// TIA Portal V19 export
FUNCTION_BLOCK "TYPIC_C301_SF_VEN"   // FB6, FBD
TITLE = TYPIC_C301_SF_VEN: Ventilator verkeerskoker
{ S7_Optimized_Access := 'TRUE' }
AUTHOR : OCOTECH
FAMILY : Typical
NAME : C301.803
// Logisch Object Besturing: C301.803
// 
// De subfunctie “ventilator verkeerskoker” verzorgt de bediening en sturing van een ventilator vanuit 3B en is tevens het raakvlak tussen 3B en de interne sturing van de ventilator.
// 
// De subfunctie kan zowel gebruikt worden voor langsventilatoren als ingangsventilatoren.
// 
// Een langsventilator heeft 2 mogelijke draairichtingen:
//  Rijrichting
//  Tegenrij
// 
// Een ingangsventilator heeft slechts 1 mogelijke draairichting:
//  Rijrichting
// 
// Deze typical werkt op dezelfde manier voor ingangsventilatoren als langsventilatoren. Bij ingangsventilatoren komen in de praktijk een aantal mogelijkheden nooit voor:
//  Op IRIS SCADA is er een andere typical voor ingangsventilatoren, deze typical heeft geen mogelijkheid voor bediening “Tegenrij”
//  Vanuit de basisfunctie wordt een cluster met ingangsventilatoren nooit in “Tegenrij” aangestuurd 
//  De waarde “Tegenrij” is nooit van toepassing voor statussen of sturingen
//  Signaleringen met betrekking tot “Tegenrij” komen nooit op
// stored: MemoryReserve 10, SetENOAutomatically false
   VAR_INPUT
      CFG_PWR { ExternalAccessible := 'False'; ExternalVisible := 'False'; ExternalWritable := 'False'} : Real;   // Vermogen ventilator
      CFG_IVEN { ExternalAccessible := 'False'; ExternalVisible := 'False'; ExternalWritable := 'False'} : USInt;   // De ventilator is een ingangsventilator
      STU_CMD_AUT { ExternalAccessible := 'False'; ExternalVisible := 'False'; ExternalWritable := 'False'} : USInt;   // Groepscommando: schakel in automatisch
      STU_ALG_LCK_SIG { ExternalAccessible := 'False'; ExternalVisible := 'False'; ExternalWritable := 'False'} : USInt;   // Onderdruk alarmen
      STU_ENE_VGV_AAN { ExternalAccessible := 'False'; ExternalVisible := 'False'; ExternalWritable := 'False'} : USInt;   // Vrijgeven of verhinderen bijschakelen energieverbruikers (verlichting / ventilatie)
   END_VAR
   VAR_OUTPUT
      VAR_VEN { ExternalAccessible := 'False'; ExternalVisible := 'False'; ExternalWritable := 'False'} : "C301_VAR_VEN_TYPIC";   // Struct met alle variabelen van de ventilator
      STU_IF_VEN { ExternalAccessible := 'False'; ExternalVisible := 'False'; ExternalWritable := 'False'} : "C301_STU_IF_VEN_TYPIC";   // Struct met alle sturingen naar de functie (IF) in de interne sturing van de ventilator
   END_VAR
   VAR_IN_OUT
      CMD : USInt;   // Sturing ventilator
      BST : USInt;   // Sturing In Dienst / Uit Dienst
      VGV_BEV : USInt;   // Vrijgave ventilator-beveiligingen onbalans en temperatuur
   END_VAR
   VAR
      BED : Struct   // Bedieningen
         ALG : Struct   // Gewenste stand
            X : "UDT_BED_ALG";
            KNOP { S7_SetPoint := 'True'} : Array[0..3] of "UDT_BED_KNOP";
         END_STRUCT;
         BST : Struct   // Bestuurbaarheid
            X : "UDT_BED_ALG";
            KNOP { S7_SetPoint := 'True'} : Array[0..1] of "UDT_BED_KNOP";
         END_STRUCT;
         RES : Struct   // Reset Storingen
            X : "UDT_BED_ALG";
            KNOP { S7_SetPoint := 'True'} : Array[0..0] of "UDT_BED_KNOP";
         END_STRUCT;
      END_STRUCT;
      BED_ALG { ExternalWritable := 'False'} : "TYPIC_HF_BED_ALG_KNOP";   // Gewenste stand
      BED_BST { ExternalWritable := 'False'} : "TYPIC_HF_BED_ALG_KNOP";   // Bestuurbaarheid
      BED_RES { ExternalWritable := 'False'} : "TYPIC_HF_BED_ALG_KNOP";   // Reset Storingen
      SIG { ExternalWritable := 'False'} : Struct   // Signaleringen
         AA01 : Bool;   // Ventilator niet bestuurbaar
         AA02 : Bool;   // Ventilator geeft storing, maar is bestuurbaar
         A001 : Bool;   // Beveiliging aangesproken
         A002 : Bool;   // Algemene storing MCC
         A003 : Bool;   // Te hoge temperatuur in de wikkelingen van de motor van de ventilator
         A004 : Bool;   // De ventilator is in onbalans
         A005 : Bool;   // Fout stroommeting fase 1
         A006 : Bool;   // Fout stroommeting fase 2
         A007 : Bool;   // Fout stroommeting fase 3
         A008 : Bool;   // Motorlade uitgeschakeld
         A009 : Bool;   // Motorlade in test
         A010 : Bool;   // Motorlade uitgereden
         A011 : Bool;   // Draadbreuk trillingsmeting
         A012 : Bool;   // Meetbereik trillingsmeting overschreden
         AT01 : Bool;   // Foute terugmelding: Motor aangestuurd, terugmelding Aan niet (of te laat) ontvangen
         AT02 : Bool;   // Foute terugmelding: Motor niet aangestuurd, terugmelding Aan blijft aanwezig
         AT03 : Bool;   // Foute terugmeldingen: terugmeldingen Positief en negatief tegelijkertijd
         M001 : Bool;   // Werkschakelaar uitgeschakeld
      END_STRUCT;
      VAR { ExternalWritable := 'False'} : Struct   // Variabelen
         TYD_TOT_AAN_UUR : USInt;   // Totaal aantal draaiuren
         ENE_MWA1 : Real;   // Stroommeting fase 1
         ENE_MWA2 : Real;   // Stroommeting fase 2
         ENE_MWA3 : Real;   // Stroommeting fase 3
         TRL_MWA : USInt;   // Trillingsmeting
         RNB : USInt;   // Reden niet bestuurbaar
         AUT : USInt;   // Beveiliging aangesproken
         VGV_SIG_VOP : Bool;   // TRUE = Signaleringen vrijgegeven voor verkeersoperator FALSE = Onderdrukt
         STS : USInt;   // Status van de ventilator
         DIR : USInt;   // Richting van de ventilator
         BMO : USInt;   // Bedieningsmode
         BST { ExternalAccessible := 'False'; ExternalVisible := 'False'} : USInt;   // Bestuurbaarheid
         PWR { ExternalAccessible := 'False'; ExternalVisible := 'False'} : Real;   // Vermogen van de ventilator
         TYD_TOT_AAN { ExternalAccessible := 'False'; ExternalVisible := 'False'} : USInt;   // Totaal aantal draaiuren
      END_STRUCT;
      HF_BST_OBS { ExternalAccessible := 'False'; ExternalVisible := 'False'; ExternalWritable := 'False'} : "TYPIC_HF_BST_OBS";   // Hulp functie besturing
   END_VAR
   // // BED.ALG.KNOP[0] : Auto
   // // BED.ALG.KNOP[1] : Rijrichting
   // // BED.ALG.KNOP[2] : Tegenrij
   // // BED.ALG.KNOP[3] : Uit
   // // BED.BST.KNOP[0] : InDienst
   // // BED.BST.KNOP[1] : UitDienst
   // // BED.RES.KNOP[0] : Reset
BEGIN

REGION Network 1: START
END_REGION

REGION Network 2: +++ Bedieningen +++
   // Vrijgave en verwerking van de bedieningen (centrale en lokale bediening). De bedienwaardes worden daarna in de verdere deelfunctionaliteiten gebruikt.
END_REGION

REGION Network 3: Knoppen BED_ALG(Gewenste stand)
   // Waardes en vrijge van de knoppen BED_ALG
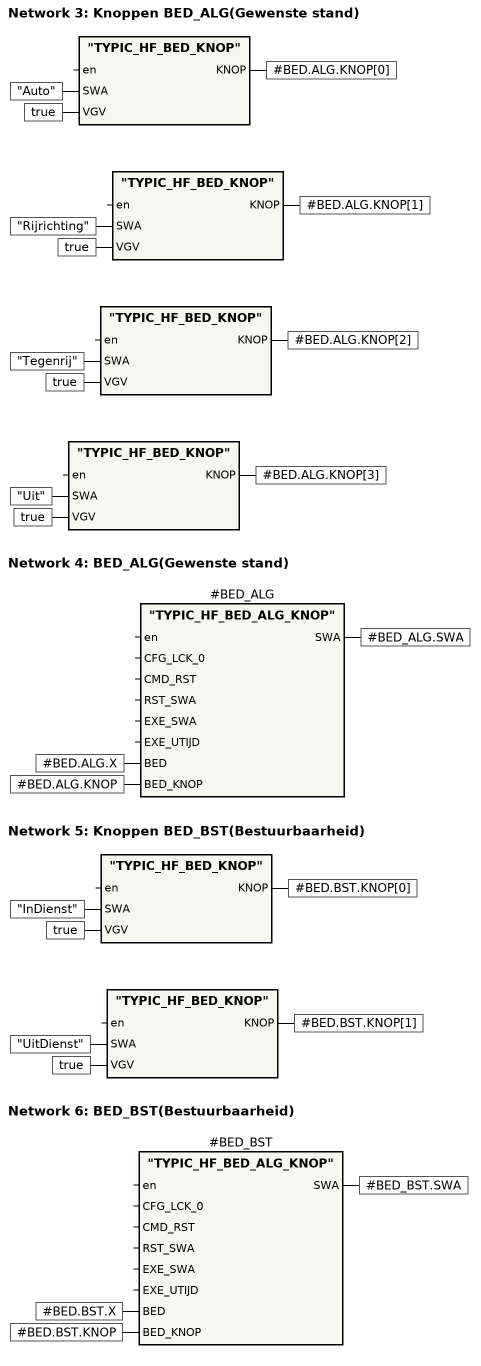
   "TYPIC_HF_BED_KNOP"(SWA := "Auto", VGV := true, KNOP => #BED.ALG.KNOP[0]);
   "TYPIC_HF_BED_KNOP"(SWA := "Rijrichting", VGV := true, KNOP => #BED.ALG.KNOP[1]);
   "TYPIC_HF_BED_KNOP"(SWA := "Tegenrij", VGV := true, KNOP => #BED.ALG.KNOP[2]);
   "TYPIC_HF_BED_KNOP"(SWA := "Uit", VGV := true, KNOP => #BED.ALG.KNOP[3]);
END_REGION

REGION Network 4: BED_ALG(Gewenste stand)
   // Verwerking BED_ALG
   #BED_ALG(BED := #BED.ALG.X, BED_KNOP := #BED.ALG.KNOP, SWA => #BED_ALG.SWA);   // "TYPIC_HF_BED_ALG_KNOP"
END_REGION

REGION Network 5: Knoppen BED_BST(Bestuurbaarheid)
   // Waardes en vrijge van de knoppen BED_BST
   "TYPIC_HF_BED_KNOP"(SWA := "InDienst", VGV := true, KNOP => #BED.BST.KNOP[0]);
   "TYPIC_HF_BED_KNOP"(SWA := "UitDienst", VGV := true, KNOP => #BED.BST.KNOP[1]);
END_REGION

REGION Network 6: BED_BST(Bestuurbaarheid)
   // Verwerking BED_BST
   #BED_BST(BED := #BED.BST.X, BED_KNOP := #BED.BST.KNOP, SWA => #BED_BST.SWA);   // "TYPIC_HF_BED_ALG_KNOP"
END_REGION

REGION Network 7: Knoppen BED_RES(Reset Storingen)
   // Waardes en vrijge van de knoppen BED_RES
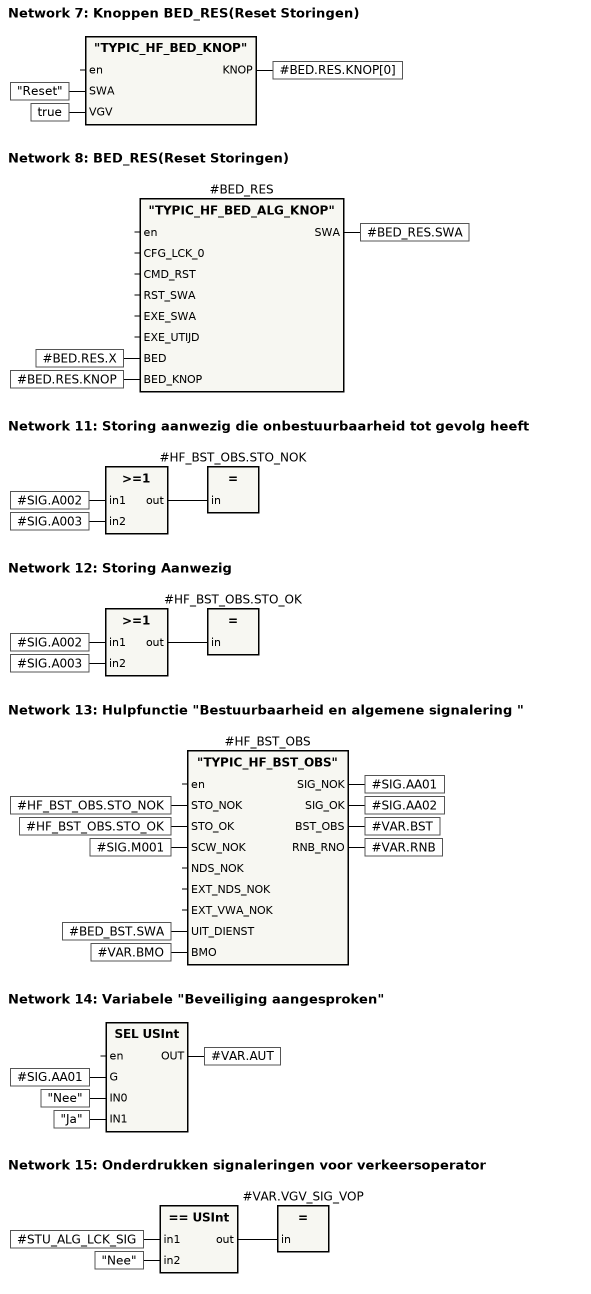
   "TYPIC_HF_BED_KNOP"(SWA := "Reset", VGV := true, KNOP => #BED.RES.KNOP[0]);
END_REGION

REGION Network 8: BED_RES(Reset Storingen)
   // Verwerking BED_RES
   #BED_RES(BED := #BED.RES.X, BED_KNOP := #BED.RES.KNOP, SWA => #BED_RES.SWA);   // "TYPIC_HF_BED_ALG_KNOP"
END_REGION

REGION Network 9: +++ Bepalen bedieningsmode +++
   // Bedieningsmode (Auto / Manueel / Hand) bepalen.
END_REGION

REGION Network 10: +++ Signaleringen en bestuurbaarheid +++
   // Aanmaken signaleringen, bepalen bestuurbaarheid (bestuurbaar / niet bestuurbaar) en bepalen reden van niet bestuurbaarheid.
END_REGION

REGION Network 11: Storing aanwezig die onbestuurbaarheid tot gevolg heeft
   // OR-verknoping van alle storingen om input STO_BST_NOK van de hulpfunctie "Bestuurbaarheid en algemene signlaring"
   #HF_BST_OBS.STO_NOK := #SIG.A002 OR #SIG.A003;
END_REGION

REGION Network 12: Storing Aanwezig
   // OR-verknoping van alle storingen om input STO_BST_OK van de hulpfunctie "Bestuurbaarheid en algemene signlaring"
   #HF_BST_OBS.STO_OK := #SIG.A002 OR #SIG.A003;
END_REGION

REGION Network 13: Hulpfunctie "Bestuurbaarheid en algemene signalering "
   // Bepalen variabele "bestuurbaarheid" en "reden niet bestuurbaar", Signaleringen "bestuurbaarheid" en "algmene storing".
   #HF_BST_OBS(STO_NOK := #HF_BST_OBS.STO_NOK,   // "TYPIC_HF_BST_OBS"
               STO_OK := #HF_BST_OBS.STO_OK,
               SCW_NOK := #SIG.M001,
               UIT_DIENST := #BED_BST.SWA,
               BMO := #VAR.BMO,
               SIG_NOK => #SIG.AA01,
               SIG_OK => #SIG.AA02,
               BST_OBS => #VAR.BST,
               RNB_RNO => #VAR.RNB);
END_REGION

REGION Network 14: Variabele "Beveiliging aangesproken"
   // De variabele VAR_AUT geef aan of er een beveilliging aangesproken is. Deze variabele laat toe dat de verkeersoperator op SCADA kan zien of er een beveilliging aangesproken is voor deze component.
   #VAR.AUT := SEL(G := #SIG.AA01, IN0 := "Nee", IN1 := "Ja");
END_REGION

REGION Network 15: Onderdrukken signaleringen voor verkeersoperator
   // Via de variabele VGV_SIG_VOP wordt aan IRIS SCADA doorgegeven of signaleringen (bestemd voor de verkeersoperator) van de deze functie zichtbaar (of onderdrukt) moeten zijn.
   #VAR.VGV_SIG_VOP := #STU_ALG_LCK_SIG = "Nee";
END_REGION

REGION Network 16: +++ Bepalen status en actueel vermogen +++
   // Status (Aan / Uit) en actueel verbruikt vermogen bepalen.
END_REGION

REGION Network 17: +++ Bepalen actuele ventilatierichting +++
   // De actuele draairichting (Uit / Rijrichting / Tegenrij) bepalen.
END_REGION

REGION Network 18: +++ Draaiuren, fasestromen en trillingsmeting +++
   // Totaal aantal draaiuren, fasestromen en trillingsmeting verwerken.
END_REGION

REGION Network 19: +++ Sturingen +++
   // Commandos naar de interne sturing van de ventilator uitsturen.
END_REGION

REGION Network 20 (SCL): EINDE
   // Variabelen van intern scada rakvlak naar outputs copieren
   #VAR_VEN.STS := #VAR.STS;
   #VAR_VEN.DIR := #VAR.DIR;
   #VAR_VEN.BMO := #VAR.BMO;
   #VAR_VEN.BST := #VAR.BST;
   #VAR_VEN.PWR := #VAR.PWR;
   #VAR_VEN.TYD_TOT_AAN := #VAR.TYD_TOT_AAN;
END_REGION
END_FUNCTION_BLOCK
